(* IEC 61131-3 sources: MXEN3002/deliverables/usb/st/test_harnesses, 5 files *)

(* ---- Test_Arm.st ---- *)
(*  Test_Arm  --  Milestones 1.5 (ROBUST FALSE) / 1.6 (ROBUST TRUE): swivel arm alone.
    Distributing I/O. go := run so the arm cycles magazine<->downstream continuously.
    FSM: 01_distributing/fsm_T1.md
*)
PROGRAM Test_Arm
VAR Panel : FB_Panel; Arm : FB_Actuator_T1; ROBUST : BOOL := FALSE; END_VAR

Panel(s1_start := Panel_S1, s2_stop := NOT Panel_S2, (* Stop wired NC *) s4_reset := Panel_S4,
      error_in := ROBUST AND Arm.error, reset_done := Arm.at_home);
Arm(run_mode := Panel.run_mode, pause_mode := Panel.pause_mode,
    reset_mode := Panel.reset_mode, error_mode := Panel.error_mode,
    sensor_home := Station_3S1, sensor_end := Station_3S2,
    go := Panel.run_mode, t_stall := T#2s, robust := ROBUST);

Station_3Y1 := Arm.valve_to_home;  // Arm_to_Magazine
Station_3Y2 := Arm.valve_to_end;   // Arm_to_Subsequent
Station_H1  := Panel.start_light;
Station_H2  := Panel.reset_light;
Panel_H4    := Panel.error_mode;   // Q2
END_PROGRAM

(* ---- Test_EjectorT2.st ---- *)
(*  Test_EjectorT2  --  Milestones 1.7 / 1.8: ejection cylinder alone.
    Distributing I/O. Stroke-completing: pause finishes the stroke to a limit.
    FSM: 01_distributing/fsm_T2.md
*)
PROGRAM Test_EjectorT2
VAR Panel : FB_Panel; Ejector : FB_Actuator_T2; ROBUST : BOOL := FALSE; END_VAR

Panel(s1_start := Panel_S1, s2_stop := NOT Panel_S2, (* Stop wired NC *) s4_reset := Panel_S4,
      error_in := ROBUST AND Ejector.error, reset_done := Ejector.at_home);
Ejector(run_mode := Panel.run_mode, pause_mode := Panel.pause_mode,
    reset_mode := Panel.reset_mode, error_mode := Panel.error_mode,
    sensor_home := Station_1B1, sensor_end := Station_1B2,
    go := Panel.run_mode, t_stall := T#2s, robust := ROBUST);

Station_1Y1 := Ejector.valve_extend;   // Magazine_Eject
Station_H1  := Panel.start_light;
Station_H2  := Panel.reset_light;
Panel_H4    := Panel.error_mode;       // Q2
END_PROGRAM

(* ---- Test_EjectorT3.st ---- *)
(*  Test_EjectorT3  --  Milestones 2.4 / 2.5: testing ejecting cylinder alone.
    Testing I/O. Single retract sensor (2B1); extended end is the stroke timer.
    Stall is caught on the retract leg. FSM: 03_testing/fsm_T3.md
*)
PROGRAM Test_EjectorT3
VAR Panel : FB_Panel; Ejector : FB_Actuator_T3; ROBUST : BOOL := FALSE; END_VAR

Panel(s1_start := Panel_S1, s2_stop := NOT Panel_S2, (* Stop wired NC *) s4_reset := Panel_S4,
      error_in := ROBUST AND Ejector.error, reset_done := Ejector.at_home);
Ejector(run_mode := Panel.run_mode, pause_mode := Panel.pause_mode,
    reset_mode := Panel.reset_mode, error_mode := Panel.error_mode,
    sensor_home := Station_2B1, go := Panel.run_mode,
    t_stroke := T#700ms, t_stall := T#2s, robust := ROBUST);

Station_2Y1 := Ejector.valve_extend;   // Advance Ejecting Cylinder
Station_H1  := Panel.start_light;
Station_H2  := Panel.reset_light;
Station_H4  := Panel.error_mode;       // Q2
END_PROGRAM

(* ---- Test_Lift.st ---- *)
(*  Test_Lift  --  Milestones 2.2 / 2.3: testing lift alone (FB_Actuator_T1 reused).
    Testing I/O. home = down (1B2/1Y1), end = up (1B1/1Y2). Switch off the air
    mid-travel to trigger the 2.3 stall. FSM: 01_distributing/fsm_T1.md
*)
PROGRAM Test_Lift
VAR Panel : FB_Panel; Lift : FB_Actuator_T1; ROBUST : BOOL := FALSE; END_VAR

Panel(s1_start := Panel_S1, s2_stop := NOT Panel_S2, (* Stop wired NC *) s4_reset := Panel_S4,
      error_in := ROBUST AND Lift.error, reset_done := Lift.at_home);
Lift(run_mode := Panel.run_mode, pause_mode := Panel.pause_mode,
    reset_mode := Panel.reset_mode, error_mode := Panel.error_mode,
    sensor_home := Station_1B2, sensor_end := Station_1B1,
    go := Panel.run_mode, t_stall := T#2s, robust := ROBUST);

Station_1Y1 := Lift.valve_to_home;  // Lift Down
Station_1Y2 := Lift.valve_to_end;   // Lift Up
Station_H1  := Panel.start_light;
Station_H2  := Panel.reset_light;
Station_H4  := Panel.error_mode;    // Q2 (testing lights are Station_H1..H4)
END_PROGRAM

(* ---- Test_Panel.st ---- *)
(*  Test_Panel  --  Milestone 1.4: control panel only, no actuators.
    Distributing I/O. reset_done := FALSE so RESET exits only on Stop, which is
    exactly what the 1.4 invalid-transition steps test. FSM: 01_distributing/fsm_panel.md
*)
PROGRAM Test_Panel
VAR Panel : FB_Panel; END_VAR

Panel(s1_start := Panel_S1, s2_stop := NOT Panel_S2, (* Stop wired NC *) s4_reset := Panel_S4,
      error_in := FALSE, reset_done := FALSE);

Station_H1 := Panel.start_light;   // start light
Station_H2 := Panel.reset_light;   // reset light
Panel_H3   := FALSE;               // Q1
Panel_H4   := Panel.error_mode;    // Q2
END_PROGRAM
